FUNCTION toErrorText : STRING(255)
VAR
	i				: INT; 
	message			: STRING(255);
	errorArray 		: ARRAY [0..5] OF ST_Event;
END_VAR

FOR i := 1 TO 5 DO
	IF GVL.lastErrorsOccurred[i].isTriggered THEN
		message := CONCAT(message, GVL.lastErrorsOccurred[i].message);
		message := CONCAT(message, ',');
	END_IF
END_FOR

toErrorText := message;

END_FUNCTION

(* stored: Version 1.1.0.1
   POU toErrorText: Id {f075bde4-1c5b-4827-acd6-3ff282e17fc7}, SpecialFunc None *)
